// TIA Portal V18 export
DATA_BLOCK "hour_min_DB_3"   // DB30
VERSION : 0.1
// stored: AutoNumber true, DBAccessibleFromOPCUA true, InstanceOfName hour_min, InstanceOfType FB
"hour_min"
   // VAR_INPUT
   //    in : Bool;
   //    reset : Bool;
   // END_VAR
   // VAR_OUTPUT
   //    outmin : Int;
   //    outhr : Int;
   // END_VAR
   // VAR RETAIN
   //    insec : Int;
   // END_VAR
   // VAR
   //    temp : Bool;
   // END_VAR
BEGIN
END_DATA_BLOCK
